FUNCTION_BLOCK ABSTRACT Component IMPLEMENTS I_Component
VAR
	_Name : T_MaxString;
	RegisteredAsComponentResult : RegistrationResult;
END_VAR

METHOD Accept
VAR_INPUT
	ComponentVisitor : I_ComponentVisitor;
END_VAR
ComponentVisitor.VisitComponent(THIS^);
END_METHOD

METHOD DeregisterWithParent
VAR_INPUT
	Parent : I_ContainComponents;
END_VAR
Parent.DeregisterComponent(THIS^);
END_METHOD

//FB_Init is always available implicitly and it is used primarily for initialization.

//The return value is not evaluated. For a specific influence, you can also declare the

//methods explicitly and provide additional code there with the standard initialization

//code. You can evaluate the return value.
METHOD FB_Init : BOOL
VAR_INPUT
	bInitRetains : BOOL; // TRUE: the retain variables are initialized (reset warm / reset cold)
	bInCopyCode	 : BOOL; // TRUE: the instance will be copied to the copy code afterward (online change)   
	Name		 : T_MaxString;
END_VAR
_Name := Name;
END_METHOD

{attribute 'monitoring' := 'call'}
PROPERTY Name : T_MaxString
GET
Name := _Name;
END_GET
SET
_Name := Name;
END_SET
END_PROPERTY

METHOD RegisterWithParent
VAR_INPUT
	Parent : I_ContainComponents;
END_VAR
RegisteredAsComponentResult := Parent.RegisterComponent(THIS^);
END_METHOD

END_FUNCTION_BLOCK

(* stored: Version 1.1.0.1, ProductVersion 3.1.4026.18
   POU Component: Id {7ca68c2e-7809-4db1-96cb-21e40a6911fb}, SpecialFunc None
   Folder Component: Id {dd63eb0a-0590-4ac7-84a0-2d1103657814}
   Folder Constructor: Id {7029559d-96b3-44f4-8e40-cfc39c228da9}
   Method Accept: Id {9a005210-45b9-436e-9e5a-8b8cb2b2ea95}
   Method DeregisterWithParent: Id {bcf6106e-efab-4aec-bbf2-ef9b6729b2d3}
   Method FB_Init: Id {5181ee6d-8a10-4110-87d4-aaf6651da738}
   Property Name: Id {34c0fc61-f2f3-4510-aa21-6e7de308a6d2}
   Get Get: Id {b36d2889-dbf5-4307-bc29-88bfde6a6b0a}
   Set Set: Id {48fdb33f-6030-41eb-a266-3d231f9f5318}
   Method RegisterWithParent: Id {41ccae3b-803b-4aef-a366-bc240eaedcd8} *)
